// TIA Portal project "2022.06.04_电机定时启动" (V17)

(* hardware
DEVICE "S7-1200 station_1"  S7-1200 Station
   slot 0: "Rack_0"  S7-1200 Rack  Rack  V1.0
   slot 1: "PLC_1"  CPU 1212C DC/DC/DC  6ES7 212-1AE40-0XB0  V4.5
*)

// ===== PLC "PLC_1"  CPU 1212C DC/DC/DC =====

VAR_GLOBAL   // PLC tag table "默认变量表"
   "启动按钮" AT %I0.0 : Bool;
   "停止按钮" AT %I0.1 : Bool;
   "电机" AT %Q0.0 : Bool;
   "中级" AT %M1.0 : Bool;
   "启动" AT %I0.2 : Bool;
   "Tag_2" AT %M1.1 : Bool;
   "电机2" AT %Q0.1 : Bool;
   "Tag_1" AT %M1.2 : Bool;
   "Tag_3" AT %Q0.2 : Bool;
END_VAR

// folder: System blocks/Program resources

DATA_BLOCK "IEC_Timer_0_DB"   // DB1
{ S7_Optimized_Access := 'TRUE' }
AUTHOR : Simatic
FAMILY : IEC
NAME : IEC_TMR
VERSION : 1.0
// stored: InstanceOfName IEC_TIMER
"IEC_TIMER"
BEGIN
END_DATA_BLOCK

DATA_BLOCK "IEC_Timer_0_DB_1"   // DB2
{ S7_Optimized_Access := 'TRUE' }
AUTHOR : Simatic
FAMILY : IEC
NAME : IEC_TMR
VERSION : 1.0
// stored: InstanceOfName IEC_TIMER
"IEC_TIMER"
BEGIN
END_DATA_BLOCK

// folder: (top level)

ORGANIZATION_BLOCK "Main"   // OB1, LAD, ProgramCycle
TITLE = "Main Program Sweep (Cycle)"
{ S7_Optimized_Access := 'TRUE' }
VERSION : 0.1
// 按下启动，5s后电机转，中级吸合起保停，按下停止按钮点击停止
   VAR_INPUT
      Initial_Call : Bool;   // Initial call of this OB
      Remanence : Bool;   // =True, if remanent data are available
   END_VAR
BEGIN

REGION Network 1
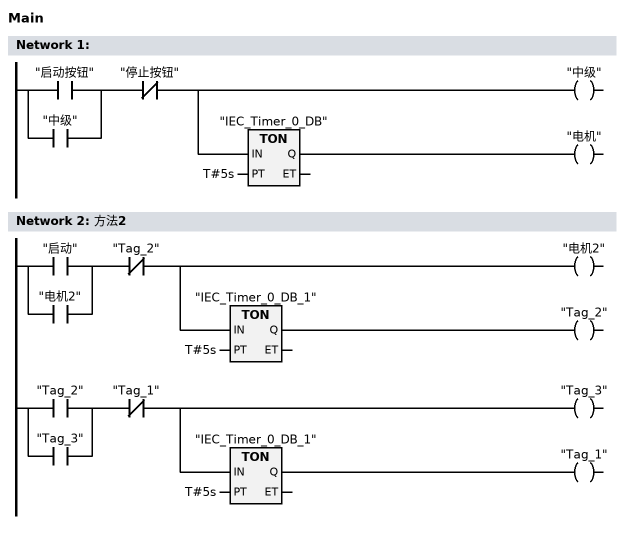
   "中级" := ("启动按钮" OR "中级") AND NOT "停止按钮";
   "IEC_Timer_0_DB".TON(IN := "中级", PT := T#5s);
   "电机" := "IEC_Timer_0_DB".Q;
END_REGION

REGION Network 2: 方法2
   "电机2" := ("启动" OR "电机2") AND NOT "Tag_2";
   "IEC_Timer_0_DB_1".TON(IN := "电机2", PT := T#5s);
   "Tag_2" := "IEC_Timer_0_DB_1".Q;
   "Tag_3" := ("Tag_2" OR "Tag_3") AND NOT "Tag_1";
   "IEC_Timer_0_DB_1".TON(IN := "Tag_3", PT := T#5s);
   "Tag_1" := "IEC_Timer_0_DB_1".Q;
END_REGION
END_ORGANIZATION_BLOCK